// Mitsubishi GX Works2 project: 拨片式分拣加叠书功能   PLC: FX2N/FX2NC

PROGRAM MAIN
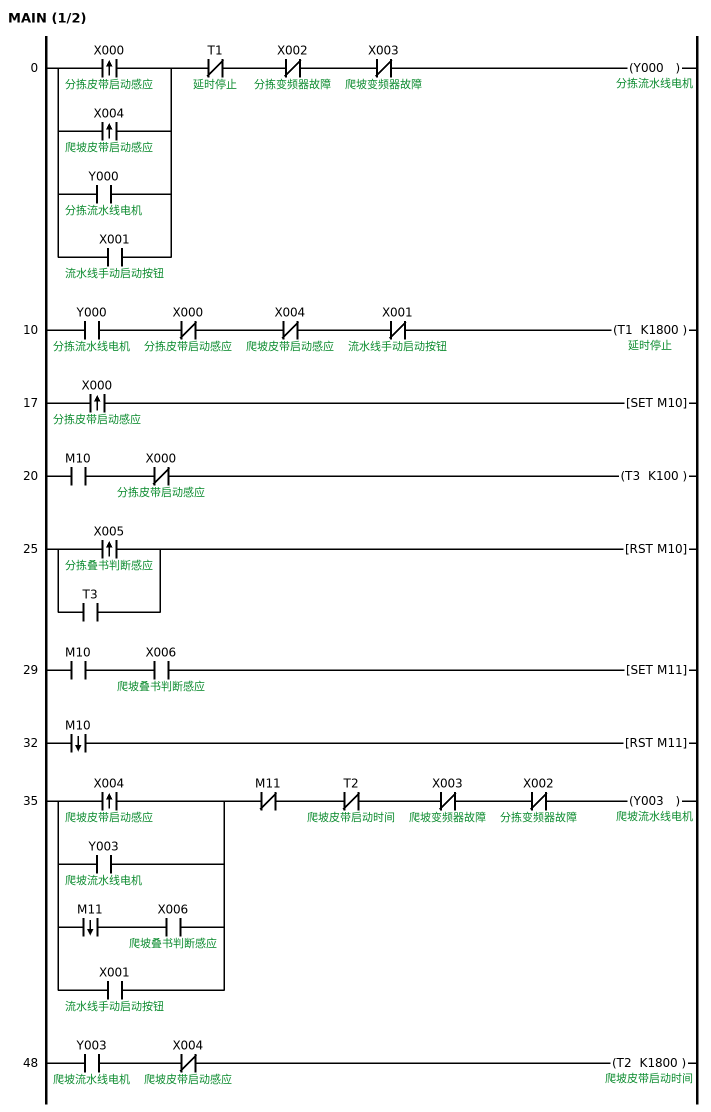
0     LDP     X000  ; 分拣皮带启动感应
      ORP     X004  ; 爬坡皮带启动感应
      OR      Y000  ; 分拣流水线电机
      OR      X001  ; 流水线手动启动按钮
      ANI     T1  ; 延时停止
      ANI     X002  ; 分拣变频器故障
      ANI     X003  ; 爬坡变频器故障
      OUT     Y000  ; 分拣流水线电机
10    LD      Y000  ; 分拣流水线电机
      ANI     X000  ; 分拣皮带启动感应
      ANI     X004  ; 爬坡皮带启动感应
      ANI     X001  ; 流水线手动启动按钮
      OUT     T1 K1800  ; 延时停止
17    LDP     X000  ; 分拣皮带启动感应
      SET     M10
20    LD      M10
      ANI     X000  ; 分拣皮带启动感应
      OUT     T3 K100
25    LDP     X005  ; 分拣叠书判断感应
      OR      T3
      RST     M10
29    LD      M10
      AND     X006  ; 爬坡叠书判断感应
      SET     M11
32    LDF     M10
      RST     M11
35    LDP     X004  ; 爬坡皮带启动感应
      OR      Y003  ; 爬坡流水线电机
      LDF     M11
      AND     X006  ; 爬坡叠书判断感应
      ORB
      OR      X001  ; 流水线手动启动按钮
      ANI     M11
      ANI     T2  ; 爬坡皮带启动时间
      ANI     X003  ; 爬坡变频器故障
      ANI     X002  ; 分拣变频器故障
      OUT     Y003  ; 爬坡流水线电机
48    LD      Y003  ; 爬坡流水线电机
      ANI     X004  ; 爬坡皮带启动感应
      OUT     T2 K1800  ; 爬坡皮带启动时间
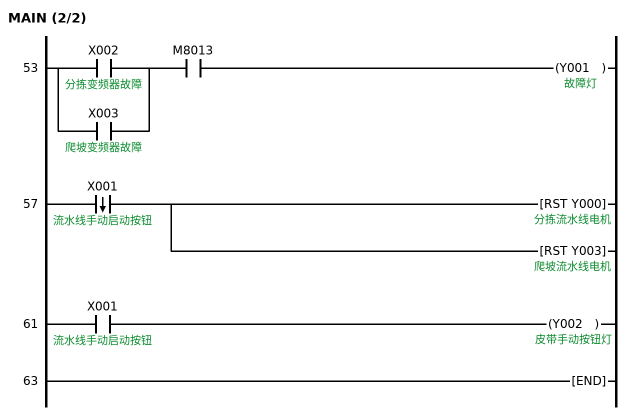
53    LD      X002  ; 分拣变频器故障
      OR      X003  ; 爬坡变频器故障
      AND     M8013
      OUT     Y001  ; 故障灯
57    LDF     X001  ; 流水线手动启动按钮
      RST     Y000  ; 分拣流水线电机
      RST     Y003  ; 爬坡流水线电机
61    LD      X001  ; 流水线手动启动按钮
      OUT     Y002  ; 皮带手动按钮灯
63    END
END_PROGRAM
